// przykalodwy program logujacy uzytkownika wizualizacji z poziomu kodu PLC
PROGRAM P_LoginFromPLC
VAR
	bLogIn 		: BOOL;
	pClient		: POINTER TO VisuElems.VisuStructClientData; 
END_VAR

IF bLogIn THEN
	VisuElems.g_ClientManager.BeginIteration(); 
	pClient := VisuElems.g_ClientManager.GetNextClient(); 
	
	WHILE pClient <> VisuElems.NULL DO 
		IF (pClient^.GlobalData.CurrentUserGroupId <> 1) THEN 
			VisuUserManagement.g_VisuUserMgmt2.LoginToUserGroup(pClient, 1, "Admin", "Administrator");
		END_IF 
		pClient := VisuElems.g_ClientManager.GetNextClient(); 
	END_WHILE
END_IF

END_PROGRAM

(* stored: Version 1.1.0.1, ProductVersion 3.1.4024.3
   POU P_LoginFromPLC: Id {6407eba1-1366-4683-b856-486fa6fb4127}, SpecialFunc None *)
